FUNCTION_BLOCK FB_Group1 EXTENDS FB_BaseGroupElement IMPLEMENTS ITF_Group1, ITF_Group1_HMI_Connector
VAR
END_VAR

END_FUNCTION_BLOCK

(* stored: Version 1.1.0.1
   POU FB_Group1: Id {dba1e16b-5cc0-0c1c-00c1-bda7f36d7e2f}, SpecialFunc None *)
